// Mitsubishi GX Works2 project: HMI 연습용 코드 1   PLC: Q03UDV

PROGRAM MAIN
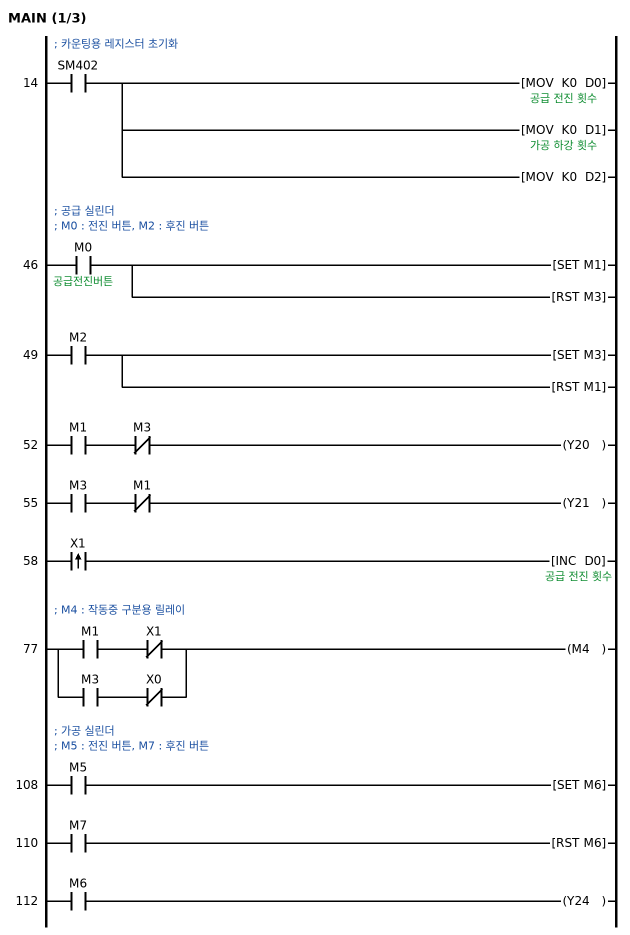
; 카운팅용 레지스터 초기화
14    LD      SM402
      MOV     K0 D0  ; 공급 전진 횟수
      MOV     K0 D1  ; 가공 하강 횟수
      MOV     K0 D2
; 공급 실린더
; M0 : 전진 버튼, M2 : 후진 버튼
46    LD      M0  ; 공급전진버튼
      SET     M1
      RST     M3
49    LD      M2
      SET     M3
      RST     M1
52    LD      M1
      ANI     M3
      OUT     Y20
55    LD      M3
      ANI     M1
      OUT     Y21
58    LDP     X1
      INC     D0
; M4 : 작동중 구분용 릴레이
77    LD      M1
      ANI     X1
      LD      M3
      ANI     X0
      ORB
      OUT     M4
; 가공 실린더
; M5 : 전진 버튼, M7 : 후진 버튼
108   LD      M5
      SET     M6
110   LD      M7
      RST     M6
112   LD      M6
      OUT     Y24
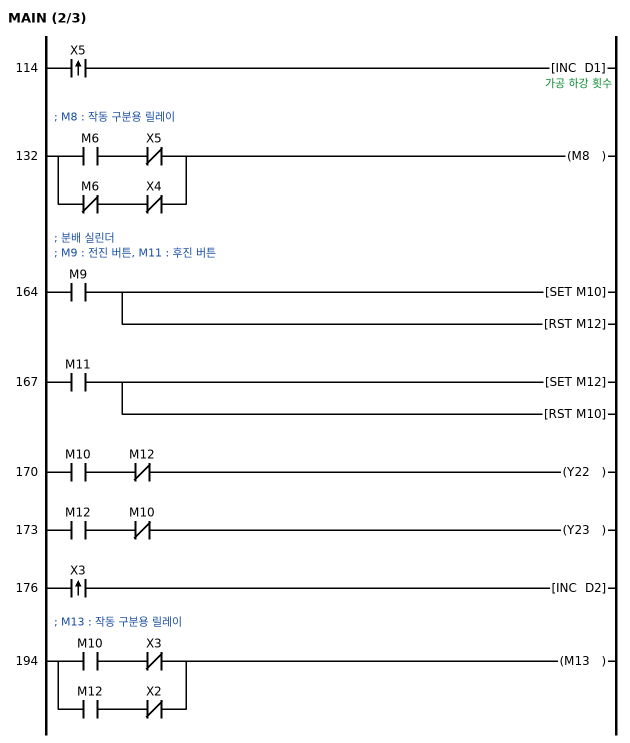
114   LDP     X5
      INC     D1
; M8 : 작동 구분용 릴레이
132   LD      M6
      ANI     X5
      LDI     M6
      ANI     X4
      ORB
      OUT     M8
; 분배 실린더
; M9 : 전진 버튼, M11 : 후진 버튼
164   LD      M9
      SET     M10
      RST     M12
167   LD      M11
      SET     M12
      RST     M10
170   LD      M10
      ANI     M12
      OUT     Y22
173   LD      M12
      ANI     M10
      OUT     Y23
176   LDP     X3
      INC     D2
; M13 : 작동 구분용 릴레이
194   LD      M10
      ANI     X3
      LD      M12
      ANI     X2
      ORB
      OUT     M13
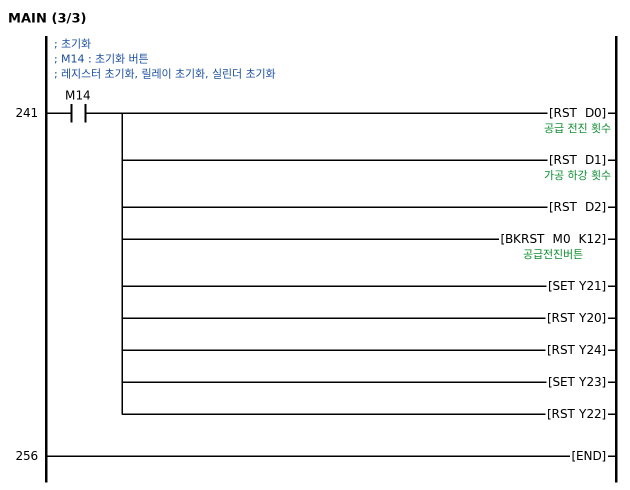
; 초기화
; M14 : 초기화 버튼
; 레지스터 초기화, 릴레이 초기화, 실린더 초기화
241   LD      M14
      RST     D0  ; 공급 전진 횟수
      RST     D1  ; 가공 하강 횟수
      RST     D2
      BKRST   M0 K12
      SET     Y21
      RST     Y20
      RST     Y24
      SET     Y23
      RST     Y22
256   END
END_PROGRAM
